FUNCTION_BLOCK TimeOfDayPointerComparer EXTENDS Object IMPLEMENTS IPointerComparer
VAR
	_ClassName : STRING := __POUNAME();
END_VAR

{attribute 'monitoring' := 'call'}
PROPERTY ClassName : STRING
GET
ClassName := _ClassName;
END_GET
END_PROPERTY

{attribute "object_name" := "Compare"}
METHOD Compare : COMPARISION_RESULT
VAR_INPUT
	left : PVOID;
	right : PVOID;
END_VAR
VAR
	leftPointer : POINTER TO TIME_OF_DAY; 
	rightPointer : POINTER TO TIME_OF_DAY; 
END_VAR
IF left = 0 AND right = 0 THEN
	Compare := COMPARISION_RESULT.FIRST_EQUAL_TO_SECOND;
	RETURN;
END_IF

IF left = 0 THEN
	Compare := COMPARISION_RESULT.FIRST_LESS_THAN_SECOND;
	RETURN;	
END_IF

IF right = 0 THEN
	Compare := COMPARISION_RESULT.FIRST_GREATER_THAN_SECOND;
	RETURN;	
END_IF

leftPointer := left;
rightPointer := right;

IF leftPointer^ < rightPointer^ THEN
	Compare := COMPARISION_RESULT.FIRST_LESS_THAN_SECOND;
ELSIF leftPointer^ > rightPointer^ THEN
	Compare := COMPARISION_RESULT.FIRST_GREATER_THAN_SECOND;
ELSE
	Compare := COMPARISION_RESULT.FIRST_EQUAL_TO_SECOND;	
END_IF
END_METHOD

{attribute 'monitoring' := 'call'}
PROPERTY Size : ULINT
GET
Size := XSIZEOF(THIS^);
END_GET
END_PROPERTY

END_FUNCTION_BLOCK

(* stored: Version 1.1.0.1
   POU TimeOfDayPointerComparer: Id {ea065f30-ce64-4029-944f-852eca6f3a7d}, SpecialFunc None
   Property ClassName: Id {ac8544c7-6138-4482-89da-ea6129e09915}
   Get Get: Id {c106ce0c-ebf9-49b8-bd12-a73358cd0ba5}
   Method Compare: Id {8e2d2050-17cd-433e-91e7-4c08b6dfd298}
   Property Size: Id {9982ca12-f65e-48e0-8ba2-2a6d8ac977ab}
   Get Get: Id {4c04bccd-ba9a-421c-9318-865960b405d3} *)
